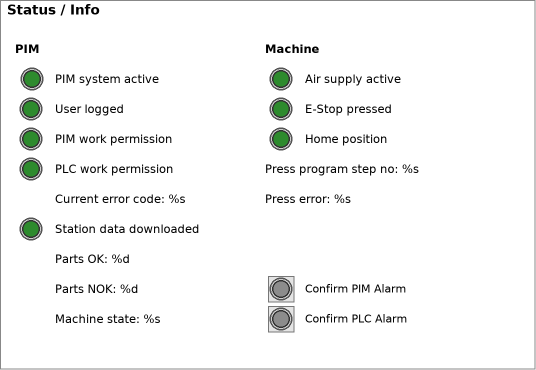
VISUALIZATION vSonicPress_SubStatus  // 536x370
VAR_IN_OUT
	fbMachine: fbSonicPress;
	fbPIM: fbPIM_Station_V3;
END_VAR
    Label (4,0 150x20), "Status / Info"
    Label (12,36 150x26), "PIM"
    Rectangle (52,96 160x26), "User logged"
    Rectangle (52,126 160x26), "PIM work permission"
    Rectangle (52,156 160x26), "PLC work permission"
    Rectangle (52,216 160x26), "Station data downloaded"
    Rectangle (52,246 160x26), "Parts OK: %d"
    Rectangle (52,276 160x26), "Parts NOK: %d"
    Rectangle (52,306 200x26), "Machine state: %s", text variable: TO_STRING(fbPIM.nMachineState)
    Label (262,36 150x26), "Machine"
    Rectangle (52,66 160x26), "PIM system active"
    Lamp1 (19,66 26x26), variable: fbPIM.stPimInOut.bPIMActive, style: Lamp-Lamp1-Green
    Lamp1 (18,96 26x26), variable: fbPIM.stPimInOut.bUserLogged, style: Lamp-Lamp1-Green
    Lamp1 (18,126 26x26), variable: NOT fbPIM.stPimInOut.bWorkBlock_PIM, style: Lamp-Lamp1-Green
    Lamp1 (18,156 26x26), variable: NOT fbPIM.stPimInOut.bWorkBlock_PLC, style: Lamp-Lamp1-Green
    Rectangle (52,186 160x26), "Current error code: %s", text variable: fbPIM.stPimInOut.sErrorCodePLC
    Lamp1 (18,216 26x26), variable: fbPIM.bStationDataOK, style: Lamp-Lamp1-Green
    Rectangle (262,186 200x26), "Press error: %s", text variable: TO_STRING(fbMachine.nError)
    Rectangle (262,156 200x26), "Press program step no: %s", text variable: fbMachine.iWorkStep
    Lamp1 (268,66 26x26), variable: fbMachine.stDigInOuts.bAirCutOffValve, style: Lamp-Lamp1-Green
    Rectangle (302,66 160x26), "Air supply active"
    Lamp1 (268,96 26x26), variable: NOT fbMachine.stDigInOuts.bSafetyStatus, style: Lamp-Lamp1-Green
    Rectangle (302,96 160x26), "E-Stop pressed"
    Lamp1 (268,126 26x26), variable: fbMachine.stDigInOuts.bHomePosSensor, style: Lamp-Lamp1-Green
    Rectangle (302,126 160x26), "Home position"
    PushSwitch (268,276 26x26), variable: fbPIM.stPimInOut.bConfirmEvent, invisible if: NOT GVL.fbUserLogin.bPermissionGranted, behaviour: TOGGLE, style: Switch-PushSwitch-Gray
    Label (302,276 150x26), "Confirm PIM Alarm", invisible if: NOT GVL.fbUserLogin.bPermissionGranted
    PushSwitch (268,306 26x26), variable: fbMachine.bServiceReset, invisible if: NOT GVL.fbUserLogin.bPermissionGranted, behaviour: TOGGLE, style: Switch-PushSwitch-Gray
    Label (302,306 150x26), "Confirm PLC Alarm", invisible if: NOT GVL.fbUserLogin.bPermissionGranted
END_VISUALIZATION

(* stored: Version 1.1.0.1, ProductVersion 3.1.4024.12
   Visu vSonicPress_SubStatus: Id {75db1514-a54b-404e-981f-648142602a51} *)
